// TIA Portal V17 export
// export: Created 2026-04-13T11:12:04.4267822Z, ExportSetting WithDefaults, DisplayName Totally Integrated Automation Portal, DisplayVersion V17 Update 4, DisplayName TIA Portal Openness, DisplayVersion V17 Update 4, DisplayName TIA Portal Version Control Interface, DisplayVersion V17, DisplayName SINAMICS Startdrive Advanced, DisplayVersion V17, DisplayName SINAMICS Startdrive G130, G150, S120, S150, SINAMICS MV, S210, DisplayVersion V17, DisplayName SINAMICS Startdrive G110M, G120, G120C, G120D, G120P, G115D, DisplayVersion V17, DisplayName STEP 7 Professional, DisplayVersion V17 Update 4, DisplayName STEP 7 Safety, DisplayVersion V17, DisplayName WinCC Professional, DisplayVersion V17 Update 4
DATA_BLOCK "YB"   // DB26
{ S7_Optimized_Access := 'TRUE' }
VERSION : 0.1
// stored: AutoNumber true, DBAccessibleFromOPCUA true, DBAccessibleFromWebserver true, IsOnlyStoredInLoadMemory false, IsRetainMemResEnabled false, IsWriteProtectedInAS false, MemoryReserve 100
   VAR
      读重量 : Real;
      A瞬时流量 : Real;
      A瞬时流速 : Real;
      A介质温度 : Real;
      A当前采集 : Real;
      A当前电流 : Real;
      A流速下限 : Real;
      A流速上限 : Real;
      A管道内径 : Real;
      B瞬时流量 : Real;
      B瞬时流速 : Real;
      B介质温度 : Real;
      B当前采集 : Real;
      B当前电流 : Real;
      B流速下限 : Real;
      B流速上限 : Real;
      B管道内径 : Real;
      秤状态 : Array[0..15] of Bool;
      秤操作 : Array[0..2] of Bool;
   END_VAR
BEGIN
END_DATA_BLOCK
